PROGRAM Calibration_1
VAR
	GVL_Calibration_Step: BOOL;
END_VAR
VAR // added by the converter: edge detectors and wires of the graphical bodies
    _w1, _w2, _w3, _w4 : BOOL;
END_VAR

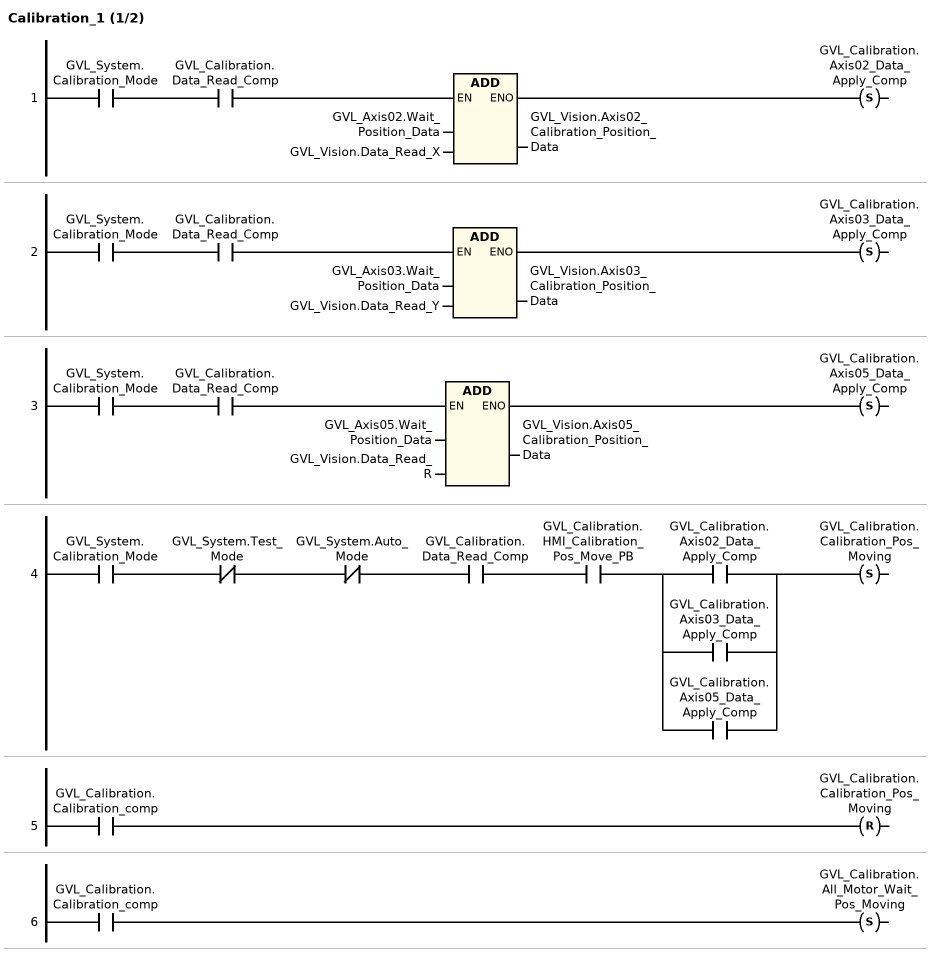
// NETWORK 1
_w1 := GVL_System.Calibration_Mode AND GVL_Calibration.Data_Read_Comp;
IF _w1 THEN
    GVL_Vision.Axis02_Calibration_Position_Data := GVL_Axis02.Wait_Position_Data + GVL_Vision.Data_Read_X;
END_IF
GVL_Calibration.Axis02_Data_Apply_Comp S= _w1;

// NETWORK 2
_w2 := GVL_System.Calibration_Mode AND GVL_Calibration.Data_Read_Comp;
IF _w2 THEN
    GVL_Vision.Axis03_Calibration_Position_Data := GVL_Axis03.Wait_Position_Data + GVL_Vision.Data_Read_Y;
END_IF
GVL_Calibration.Axis03_Data_Apply_Comp S= _w2;

// NETWORK 3
_w3 := GVL_System.Calibration_Mode AND GVL_Calibration.Data_Read_Comp;
IF _w3 THEN
    GVL_Vision.Axis05_Calibration_Position_Data := GVL_Axis05.Wait_Position_Data + GVL_Vision.Data_Read_R;
END_IF
GVL_Calibration.Axis05_Data_Apply_Comp S= _w3;

// NETWORK 4
GVL_Calibration.Calibration_Pos_Moving S= GVL_System.Calibration_Mode AND NOT GVL_System.Test_Mode AND NOT GVL_System.Auto_Mode AND GVL_Calibration.Data_Read_Comp AND GVL_Calibration.HMI_Calibration_Pos_Move_PB AND (GVL_Calibration.Axis02_Data_Apply_Comp OR GVL_Calibration.Axis03_Data_Apply_Comp OR GVL_Calibration.Axis05_Data_Apply_Comp);

// NETWORK 5
GVL_Calibration.Calibration_Pos_Moving R= GVL_Calibration.Calibration_comp;

// NETWORK 6
GVL_Calibration.All_Motor_Wait_Pos_Moving S= GVL_Calibration.Calibration_comp;

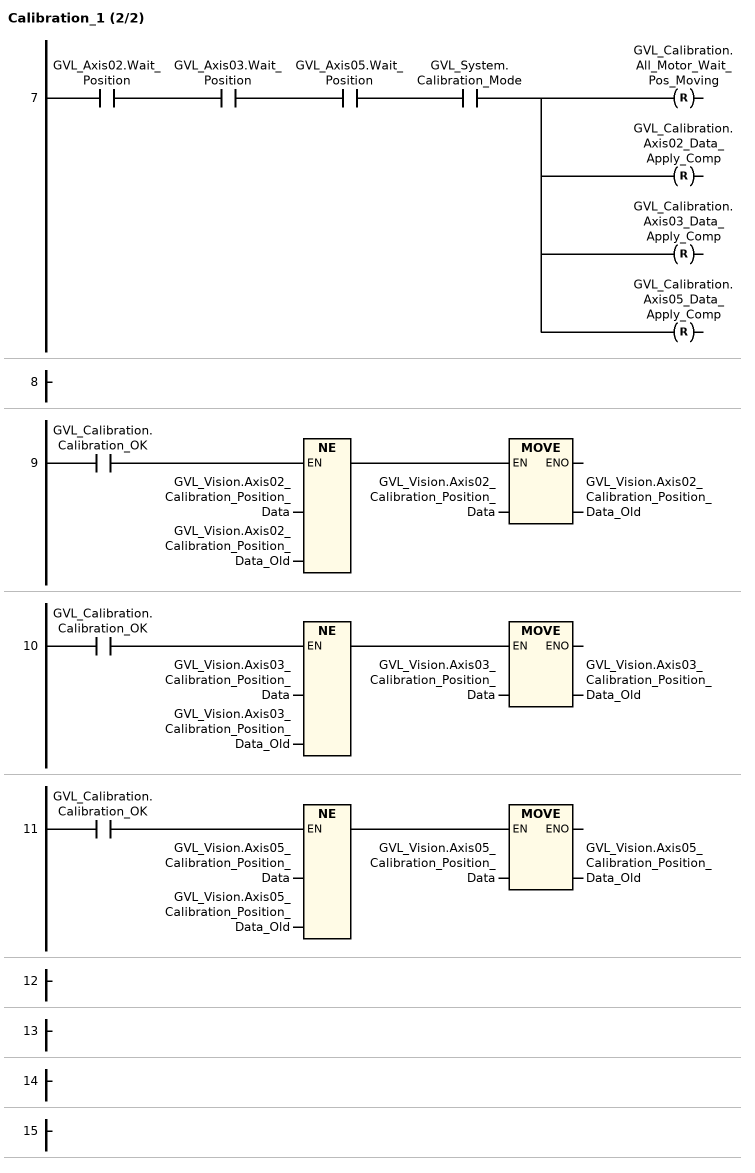
// NETWORK 7
_w4 := GVL_Axis02.Wait_Position AND GVL_Axis03.Wait_Position AND GVL_Axis05.Wait_Position AND GVL_System.Calibration_Mode;
GVL_Calibration.All_Motor_Wait_Pos_Moving R= _w4;
GVL_Calibration.Axis02_Data_Apply_Comp R= _w4;
GVL_Calibration.Axis03_Data_Apply_Comp R= _w4;
GVL_Calibration.Axis05_Data_Apply_Comp R= _w4;

// NETWORK 8

// NETWORK 9
IF GVL_Calibration.Calibration_OK AND GVL_Vision.Axis02_Calibration_Position_Data <> GVL_Vision.Axis02_Calibration_Position_Data_Old THEN
    GVL_Vision.Axis02_Calibration_Position_Data_Old := GVL_Vision.Axis02_Calibration_Position_Data;
END_IF

// NETWORK 10
IF GVL_Calibration.Calibration_OK AND GVL_Vision.Axis03_Calibration_Position_Data <> GVL_Vision.Axis03_Calibration_Position_Data_Old THEN
    GVL_Vision.Axis03_Calibration_Position_Data_Old := GVL_Vision.Axis03_Calibration_Position_Data;
END_IF

// NETWORK 11
IF GVL_Calibration.Calibration_OK AND GVL_Vision.Axis05_Calibration_Position_Data <> GVL_Vision.Axis05_Calibration_Position_Data_Old THEN
    GVL_Vision.Axis05_Calibration_Position_Data_Old := GVL_Vision.Axis05_Calibration_Position_Data;
END_IF

// NETWORK 12

// NETWORK 13

// NETWORK 14

// NETWORK 15

END_PROGRAM

(* stored: Version 1.1.0.1, ProductVersion 3.1.4024.15
   POU Calibration_1: Id {fdbd1f73-1447-463e-a0d1-f5befde9fc62}, SpecialFunc None *)
